FUNCTION_BLOCK FB_PetrolEngine

VAR
	nEngineCc : INT;
	fConsumption : REAL := 20;
END_VAR

END_FUNCTION_BLOCK

(* stored: Version 1.1.0.1, ProductVersion 3.1.4024.16
   POU FB_PetrolEngine: Id {d8e33b41-3fcf-4f3f-9526-e4217ebe6887}, SpecialFunc None *)
